# EPICS substitutions: slacApp/Db/IOCNAME-pattern.substitutions
#
# Pattern records
file evrPatternAll.db
{
#           Device        ,SLC Pattern  EVR/Trigger
#                          Check LNK      Links
  pattern { DEVICE        ,  LINK4    , LINK5, LINK6, TREF   , TS1ST, TS2ND}
#          { IOCNAME ,   ""      ,  ""  ,  ""  , 1.03E06,   3  ,   6  }
           { IOCNAME ,   ""      ,  ""  ,  ""  , 1.03E06,   1  ,   4  }
}
# Event records
file evrEventAll.db
{
  pattern { DEVICE   }
          { IOCNAME}
}
